{attribute 'pack_mode' := '1'}
TYPE TRobotPos :
STRUCT
	X		: LREAL;
	Y		: LREAL;
	Z		: LREAL;
	Theta	: LREAL;
END_STRUCT
END_TYPE

(* stored: Version 1.1.0.1, ProductVersion 3.1.4022.12
   DUT TRobotPos: Id {fd829643-43d3-4ace-82d3-f7c317b3b83a} *)
